(* PLC project LD_TEST, Beremiz BREMIZ 1 *)
(* stored: contentDescription This tests LD language, companyURL www.beremiz.org, productRelease 1, creationDateTime 2007-07-07 11:58:26 *)

PROGRAM MAIN_TEST
  VAR
    QX1 AT %QX1 : BOOL;
    QX2 AT %QX2 : BOOL;
    QX3 AT %QX3 : BOOL;
    IX1 AT %IX1 : BOOL;
    IX2 AT %IX2 : BOOL;
    IX3 AT %IX3 : BOOL;
  END_VAR

(* LD diagram, written out as Structured Text *)
END_PROGRAM

CONFIGURATION STD_CONF
  RESOURCE STD_RESSOURCE ON PLC
    TASK STD_TASK(INTERVAL := 00:00:00.100000, PRIORITY := 0);
    PROGRAM MAIN_INSTANCE : MAIN_TEST;
  END_RESOURCE
END_CONFIGURATION
